(* Logix 5000 project; controller Sucrose_Main Emulate 5570 rev 20.12; software revision 20.01; part 6 of 30 *)
(* tags used below, declared in another part *)
   Alarm_ACK_Master_Timer : TIMER;
   DI_E20_1 : ALIAS FOR FLX_E20:1:I;   // Discrete Input EN2T_FLX 192.168.1.20
   DI_E23_5 : ALIAS FOR FLX_E23:5:I;   // Discrete Input EN2T_FLX 192.168.1.23
   DO_E20_5 : ALIAS FOR FLX_E20:5:O;   // Discrete Output EN2T_FLX 192.168.1.20
   DO_E20_6 : ALIAS FOR FLX_E20:6:O;   // Discrete Output EN2T_FLX 192.168.1.20
   DO_E24_1 : ALIAS FOR FLX_E24:1:O;   // Discrete Output EN2T_FLX 192.168.1.24
   FV610101_AOI : QSI_Flow_Valve;   // FV-61-01-01-O CIP SUPPLY TO SUCROSE TANK #1 VALVE OPEN
   FV610201_AOI : QSI_Flow_Valve;   // FV-61-02-01-O CIP SUPPLY TO SUCROSE TANK #2 VALVE OPEN
   FV610301_AOI : QSI_Flow_Valve;   // FV-61-03-01-O CIP SUPPLY TO SUCROSE TANK #3 VALVE OPEN
   FV610411_AOI : QSI_Flow_Valve;   // FV-61-04-11 CIP SUPPLY TO TRANSFER PUMP #1 OR TO DRAIN DIVERT VALVE
   FV610412_AOI : QSI_Flow_Valve;   // FV-61-04-12 CIP SUPPLY TO TRANSFER PUMP #2 OR TO DRAIN DIVERT VALVE
   FV620301_AOI : QSI_Flow_Valve;   // FV-62-03-01-O SUCROSE TANK #3 TO CIP RETURN PUMP MIX PROOF VALVE OPEN
   FV620400_AOI : QSI_Flow_Valve;   // FV-62-04-00 CIP RETURN LOW POINT DRAIN VALVE
   FV620401_AOI : QSI_Flow_Valve;   // FV-62-04-01-O CIP RETURN PUMP #1 TO FILTER SYSTEM MIX PROOF VALVE OPEN
   FV620402_AOI : QSI_Flow_Valve;   // FV-62-04-02-O CIP RETURN PUMP #2 TO FILTER SYSTEM MIX PROOF VALVE OPEN
   Sucrose_MM_Enable : BOOL;
   SucroseCIP_P230401_REMOTE : CIP_REMOTE;
   SucroseCIP_P230402_REMOTE : CIP_REMOTE;
   SucroseCIP_TK230101_REMOTE : CIP_REMOTE;
   SucroseCIP_TK230201_REMOTE : CIP_REMOTE;
   SucroseCIP_TK230301_REMOTE : CIP_REMOTE;
   SucroseTanks : Area_Program;
(* CIP_RemoteArea_EN2T_IO_Discrete_DO_E20_5, continued *)

ROUTINE _03_FV620301   (* ladder *)
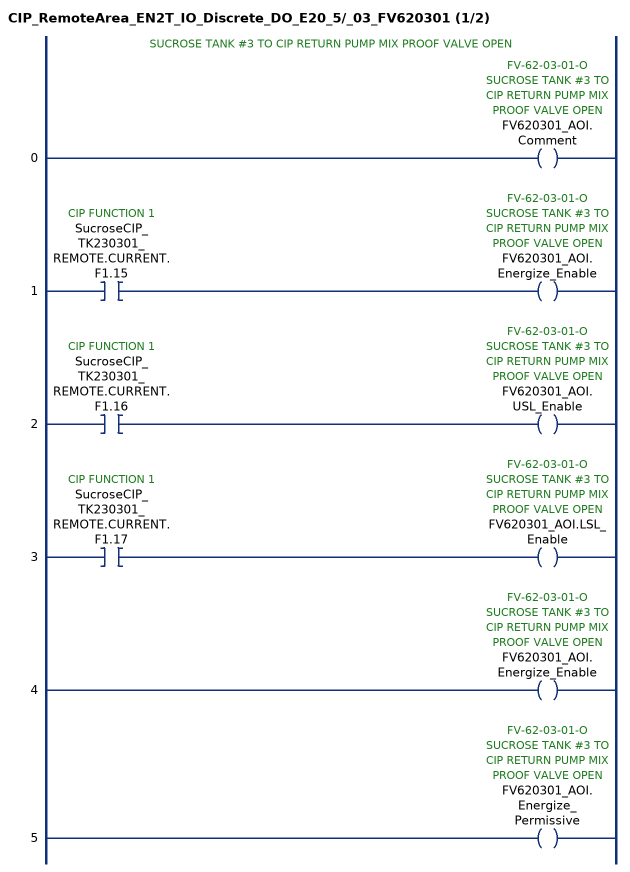
   // SUCROSE TANK #3 TO CIP RETURN PUMP MIX PROOF VALVE OPEN
   0: OTE(FV620301_AOI.Comment);
   1: XIC(SucroseCIP_TK230301_REMOTE.CURRENT.F1.15)OTE(FV620301_AOI.Energize_Enable);
   2: XIC(SucroseCIP_TK230301_REMOTE.CURRENT.F1.16)OTE(FV620301_AOI.USL_Enable);
   3: XIC(SucroseCIP_TK230301_REMOTE.CURRENT.F1.17)OTE(FV620301_AOI.LSL_Enable);
   4: OTE(FV620301_AOI.Energize_Enable);
   5: OTE(FV620301_AOI.Energize_Permissive);
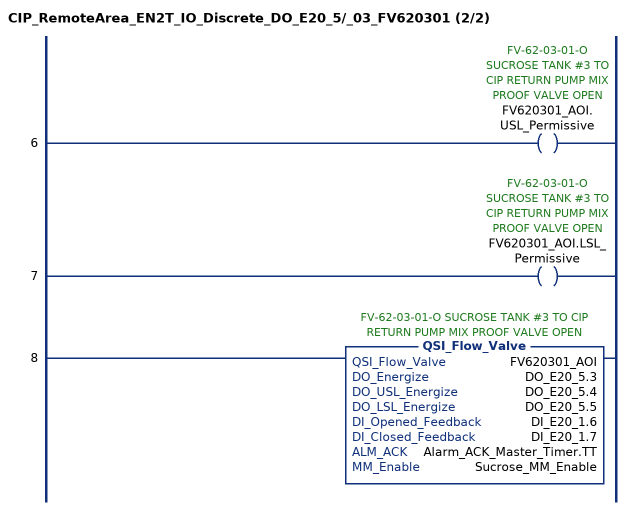
   6: OTE(FV620301_AOI.USL_Permissive);
   7: OTE(FV620301_AOI.LSL_Permissive);
   8: QSI_Flow_Valve(FV620301_AOI,DO_E20_5.3,DO_E20_5.4,DO_E20_5.5,DI_E20_1.6,DI_E20_1.7,Alarm_ACK_Master_Timer.TT,Sucrose_MM_Enable);
END_ROUTINE

ROUTINE _06_FV620401   (* ladder *)
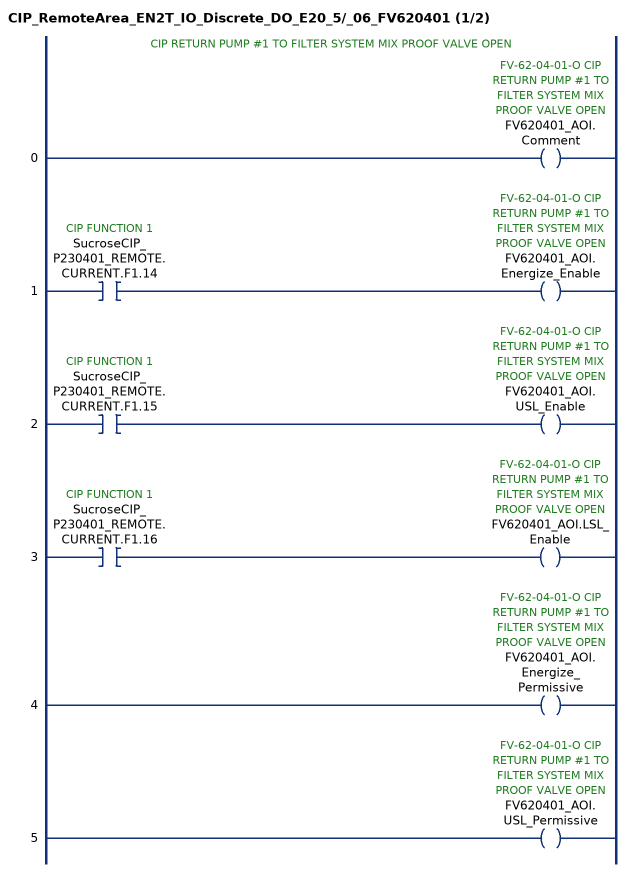
   // CIP RETURN PUMP #1 TO FILTER SYSTEM MIX PROOF VALVE OPEN
   0: OTE(FV620401_AOI.Comment);
   1: XIC(SucroseCIP_P230401_REMOTE.CURRENT.F1.14)OTE(FV620401_AOI.Energize_Enable);
   2: XIC(SucroseCIP_P230401_REMOTE.CURRENT.F1.15)OTE(FV620401_AOI.USL_Enable);
   3: XIC(SucroseCIP_P230401_REMOTE.CURRENT.F1.16)OTE(FV620401_AOI.LSL_Enable);
   4: OTE(FV620401_AOI.Energize_Permissive);
   5: OTE(FV620401_AOI.USL_Permissive);
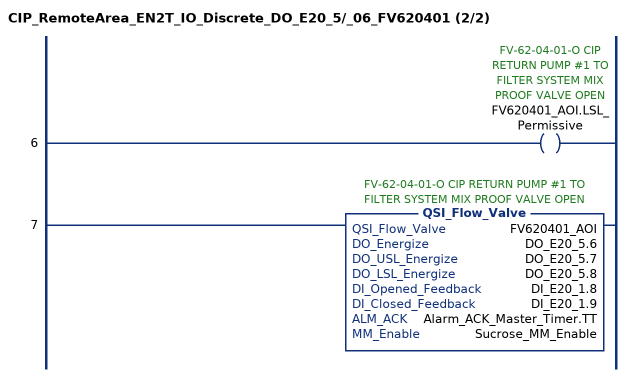
   6: OTE(FV620401_AOI.LSL_Permissive);
   7: QSI_Flow_Valve(FV620401_AOI,DO_E20_5.6,DO_E20_5.7,DO_E20_5.8,DI_E20_1.8,DI_E20_1.9,Alarm_ACK_Master_Timer.TT,Sucrose_MM_Enable);
END_ROUTINE

ROUTINE _09_FV620402   (* ladder *)
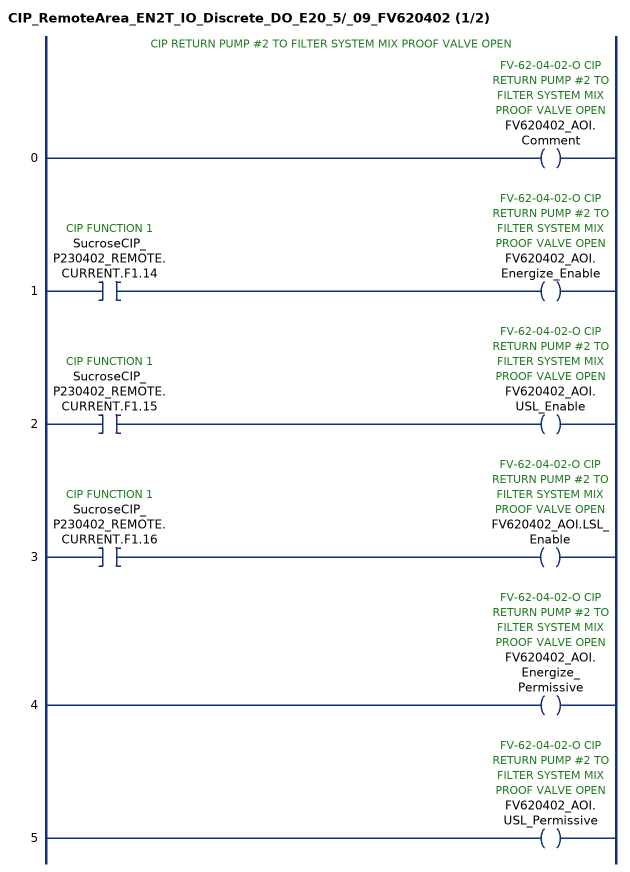
   // CIP RETURN PUMP #2 TO FILTER SYSTEM MIX PROOF VALVE OPEN
   0: OTE(FV620402_AOI.Comment);
   1: XIC(SucroseCIP_P230402_REMOTE.CURRENT.F1.14)OTE(FV620402_AOI.Energize_Enable);
   2: XIC(SucroseCIP_P230402_REMOTE.CURRENT.F1.15)OTE(FV620402_AOI.USL_Enable);
   3: XIC(SucroseCIP_P230402_REMOTE.CURRENT.F1.16)OTE(FV620402_AOI.LSL_Enable);
   4: OTE(FV620402_AOI.Energize_Permissive);
   5: OTE(FV620402_AOI.USL_Permissive);
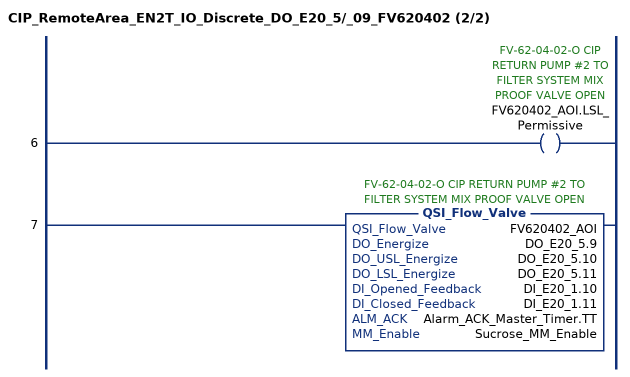
   6: OTE(FV620402_AOI.LSL_Permissive);
   7: QSI_Flow_Valve(FV620402_AOI,DO_E20_5.9,DO_E20_5.10,DO_E20_5.11,DI_E20_1.10,DI_E20_1.11,Alarm_ACK_Master_Timer.TT,Sucrose_MM_Enable);
END_ROUTINE

ROUTINE MainRoutine   (* ladder *)
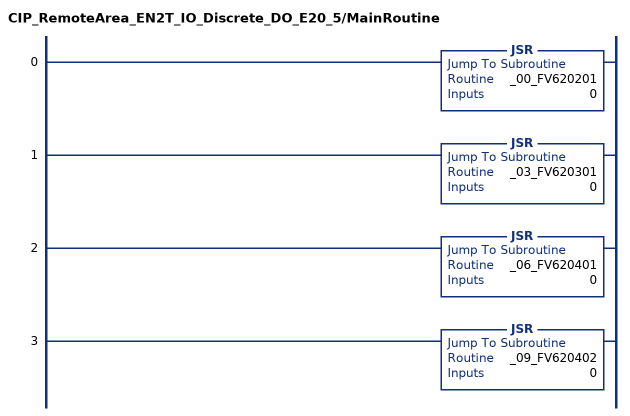
   0: JSR(_00_FV620201,0);
   1: JSR(_03_FV620301,0);
   2: JSR(_06_FV620401,0);
   3: JSR(_09_FV620402,0);
END_ROUTINE
END_PROGRAM

PROGRAM CIP_RemoteArea_EN2T_IO_Discrete_DO_E20_6   (* main routine MainRoutine *)

ROUTINE _02_FV610411   (* ladder *)
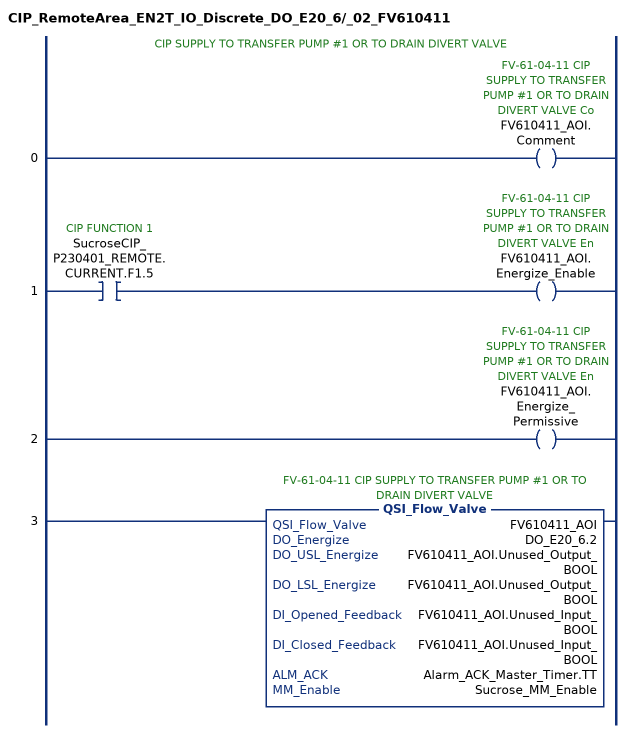
   // CIP SUPPLY TO TRANSFER PUMP #1 OR TO DRAIN DIVERT VALVE
   0: OTE(FV610411_AOI.Comment);
   1: XIC(SucroseCIP_P230401_REMOTE.CURRENT.F1.5)OTE(FV610411_AOI.Energize_Enable);
   2: OTE(FV610411_AOI.Energize_Permissive);
   3: QSI_Flow_Valve(FV610411_AOI,DO_E20_6.2,FV610411_AOI.Unused_Output_BOOL,FV610411_AOI.Unused_Output_BOOL,FV610411_AOI.Unused_Input_BOOL,FV610411_AOI.Unused_Input_BOOL,Alarm_ACK_Master_Timer.TT,Sucrose_MM_Enable);
END_ROUTINE

ROUTINE _03_FV610412   (* ladder *)
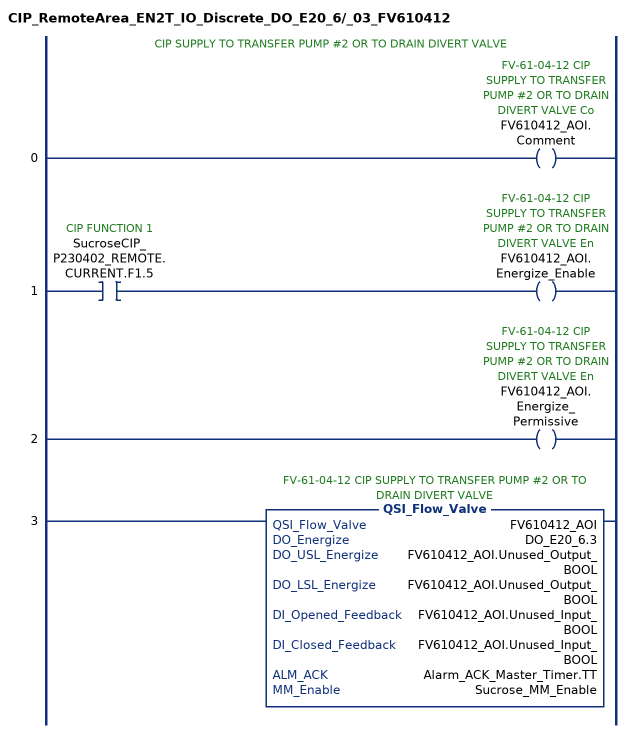
   // CIP SUPPLY TO TRANSFER PUMP #2 OR TO DRAIN DIVERT VALVE
   0: OTE(FV610412_AOI.Comment);
   1: XIC(SucroseCIP_P230402_REMOTE.CURRENT.F1.5)OTE(FV610412_AOI.Energize_Enable);
   2: OTE(FV610412_AOI.Energize_Permissive);
   3: QSI_Flow_Valve(FV610412_AOI,DO_E20_6.3,FV610412_AOI.Unused_Output_BOOL,FV610412_AOI.Unused_Output_BOOL,FV610412_AOI.Unused_Input_BOOL,FV610412_AOI.Unused_Input_BOOL,Alarm_ACK_Master_Timer.TT,Sucrose_MM_Enable);
END_ROUTINE

ROUTINE _07_FV620400   (* ladder *)
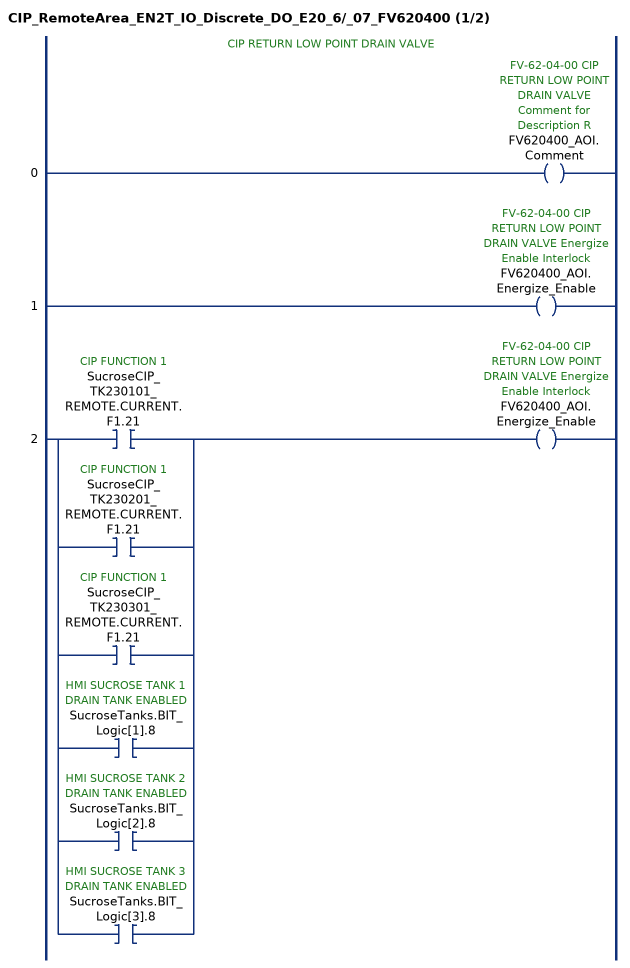
   // CIP RETURN LOW POINT DRAIN VALVE
   0: OTE(FV620400_AOI.Comment);
   1: OTE(FV620400_AOI.Energize_Enable);
   2: [XIC(SucroseCIP_TK230101_REMOTE.CURRENT.F1.21) ,XIC(SucroseCIP_TK230201_REMOTE.CURRENT.F1.21) ,XIC(SucroseCIP_TK230301_REMOTE.CURRENT.F1.21) ,XIC(SucroseTanks.BIT_Logic[1].8) ,XIC(SucroseTanks.BIT_Logic[2].8) ,XIC(SucroseTanks.BIT_Logic[3].8) ]OTE(FV620400_AOI.Energize_Enable);
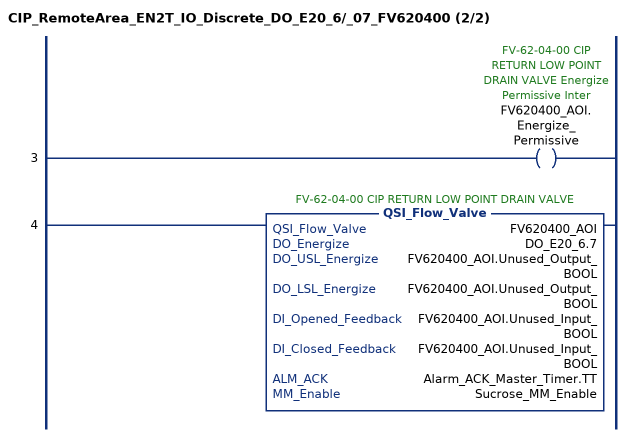
   3: OTE(FV620400_AOI.Energize_Permissive);
   4: QSI_Flow_Valve(FV620400_AOI,DO_E20_6.7,FV620400_AOI.Unused_Output_BOOL,FV620400_AOI.Unused_Output_BOOL,FV620400_AOI.Unused_Input_BOOL,FV620400_AOI.Unused_Input_BOOL,Alarm_ACK_Master_Timer.TT,Sucrose_MM_Enable);
END_ROUTINE

ROUTINE MainRoutine   (* ladder *)
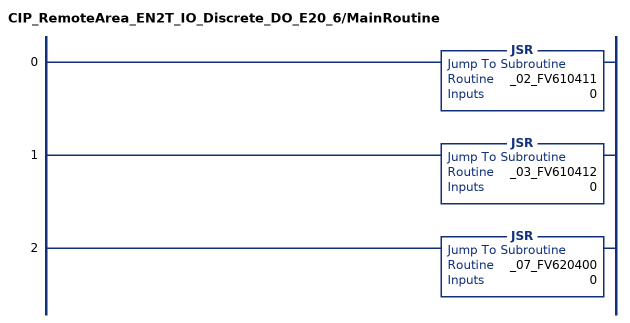
   0: JSR(_02_FV610411,0);
   1: JSR(_03_FV610412,0);
   2: JSR(_07_FV620400,0);
END_ROUTINE
END_PROGRAM

PROGRAM CIP_RemoteArea_EN2T_IO_Discrete_DO_E24_1   (* main routine MainRoutine *)

ROUTINE _06_FV610101   (* ladder *)
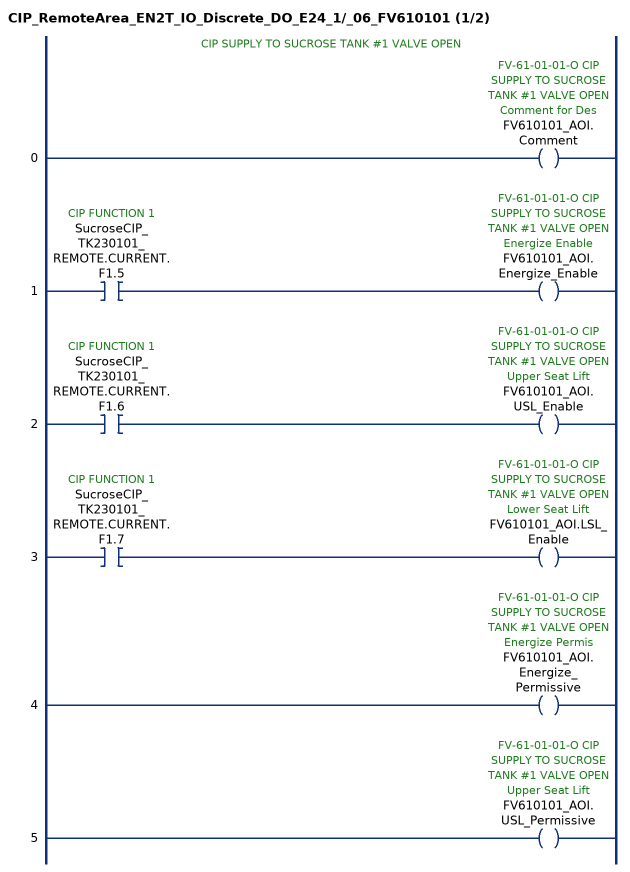
   // CIP SUPPLY TO SUCROSE TANK #1 VALVE OPEN
   0: OTE(FV610101_AOI.Comment);
   1: XIC(SucroseCIP_TK230101_REMOTE.CURRENT.F1.5)OTE(FV610101_AOI.Energize_Enable);
   2: XIC(SucroseCIP_TK230101_REMOTE.CURRENT.F1.6)OTE(FV610101_AOI.USL_Enable);
   3: XIC(SucroseCIP_TK230101_REMOTE.CURRENT.F1.7)OTE(FV610101_AOI.LSL_Enable);
   4: OTE(FV610101_AOI.Energize_Permissive);
   5: OTE(FV610101_AOI.USL_Permissive);
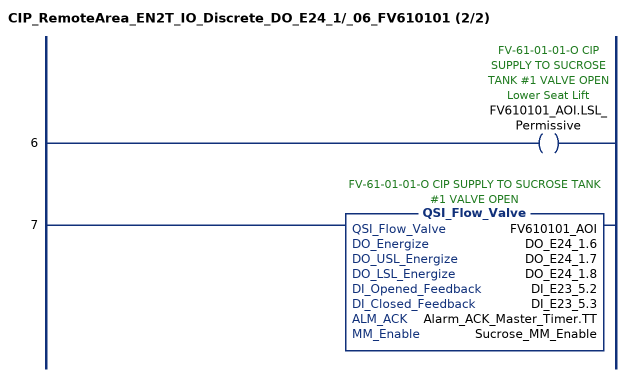
   6: OTE(FV610101_AOI.LSL_Permissive);
   7: QSI_Flow_Valve(FV610101_AOI,DO_E24_1.6,DO_E24_1.7,DO_E24_1.8,DI_E23_5.2,DI_E23_5.3,Alarm_ACK_Master_Timer.TT,Sucrose_MM_Enable);
END_ROUTINE

ROUTINE _09_FV610201   (* ladder *)
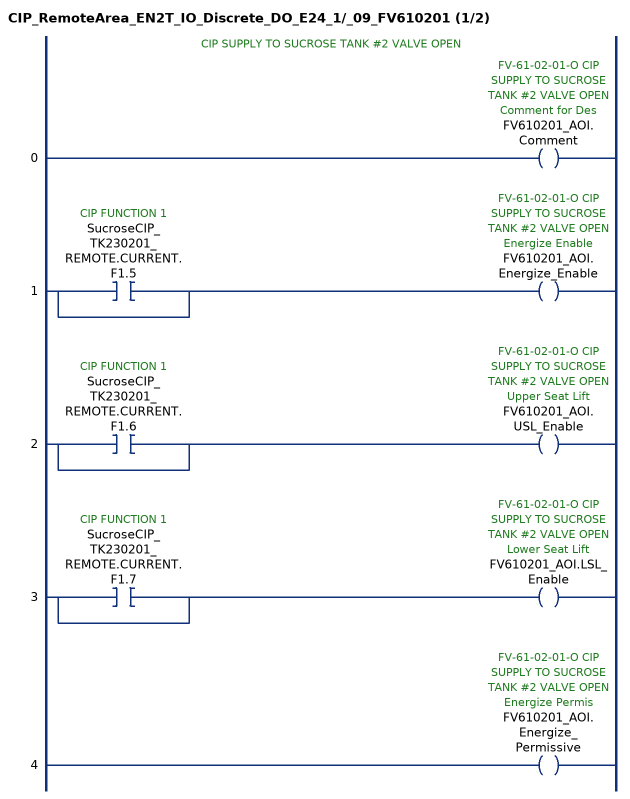
   // CIP SUPPLY TO SUCROSE TANK #2 VALVE OPEN
   0: OTE(FV610201_AOI.Comment);
   1: [XIC(SucroseCIP_TK230201_REMOTE.CURRENT.F1.5) ,]OTE(FV610201_AOI.Energize_Enable);
   2: [XIC(SucroseCIP_TK230201_REMOTE.CURRENT.F1.6) ,]OTE(FV610201_AOI.USL_Enable);
   3: [XIC(SucroseCIP_TK230201_REMOTE.CURRENT.F1.7) ,]OTE(FV610201_AOI.LSL_Enable);
   4: OTE(FV610201_AOI.Energize_Permissive);
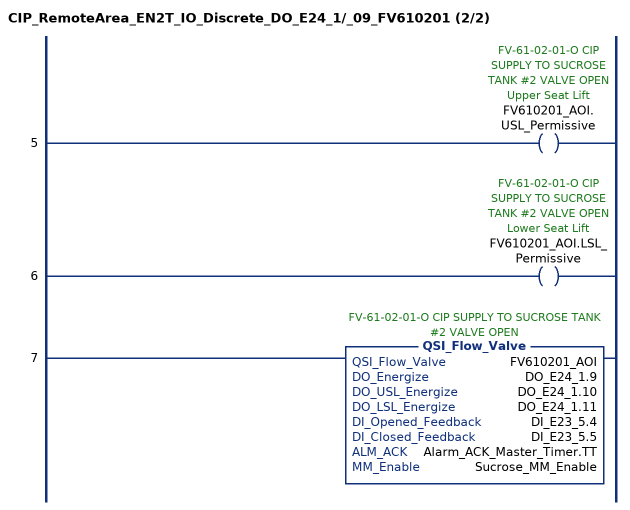
   5: OTE(FV610201_AOI.USL_Permissive);
   6: OTE(FV610201_AOI.LSL_Permissive);
   7: QSI_Flow_Valve(FV610201_AOI,DO_E24_1.9,DO_E24_1.10,DO_E24_1.11,DI_E23_5.4,DI_E23_5.5,Alarm_ACK_Master_Timer.TT,Sucrose_MM_Enable);
END_ROUTINE

ROUTINE _12_FV610301   (* ladder *)
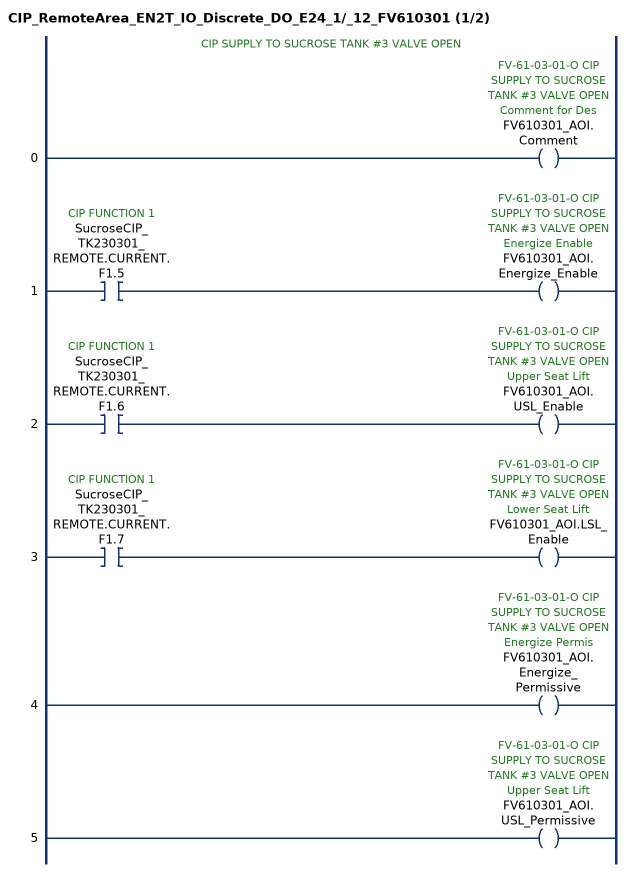
   // CIP SUPPLY TO SUCROSE TANK #3 VALVE OPEN
   0: OTE(FV610301_AOI.Comment);
   1: XIC(SucroseCIP_TK230301_REMOTE.CURRENT.F1.5)OTE(FV610301_AOI.Energize_Enable);
   2: XIC(SucroseCIP_TK230301_REMOTE.CURRENT.F1.6)OTE(FV610301_AOI.USL_Enable);
   3: XIC(SucroseCIP_TK230301_REMOTE.CURRENT.F1.7)OTE(FV610301_AOI.LSL_Enable);
   4: OTE(FV610301_AOI.Energize_Permissive);
   5: OTE(FV610301_AOI.USL_Permissive);
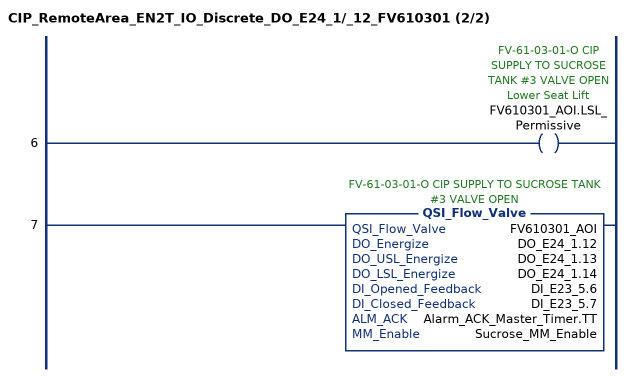
   6: OTE(FV610301_AOI.LSL_Permissive);
   7: QSI_Flow_Valve(FV610301_AOI,DO_E24_1.12,DO_E24_1.13,DO_E24_1.14,DI_E23_5.6,DI_E23_5.7,Alarm_ACK_Master_Timer.TT,Sucrose_MM_Enable);
END_ROUTINE
